TEXTLIST AUTOMATA_lepesek2
  0 = 'Készenléti állapot'
  1 = 'A szán indítása'
  3 = '6. hegesztés, várakozás a szánra'
  4 = '6. hegesztés, fej indítása'
  5 = '6. hegesztés, várakozás a fejre'
  6 = '6. hegesztés, hegesztés folyamatban'
  7 = '6. hegesztés, fej vissza'
  8 = '6. hegesztés, fej vissza'
  9 = 'A szán indítása'
  11 = '7. hegesztés, várakozás a szánra'
  12 = '7. hegesztés, fej indítása'
  13 = '7. hegesztés, várakozás a fejre'
  14 = '7. hegesztés, hegesztés folyamatban'
  15 = '7. hegesztés, fej vissza'
  16 = '7. hegesztés, fej vissza'
  17 = 'A szán indítása'
  18 = 'Kappe felhelyezés, várakozás a szánra'
  19 = 'Várakozás a robotra'
  20 = 'A robot eredmény törlésére vár'
  21 = 'A robot felhelyezi a kappét'
  22 = 'A szán indítása'
  23 = 'Kappe rögzítés, várakozás a szánra'
  24 = 'Kappe rögzítés indítása'
  27 = 'Várakozás a kappe rögzítés végére'
  28 = 'Mérés, várakozás a szánra'
  29 = 'Mérésválasztás'
  30 = 'Várakozás a mérés végére'
  31 = 'Lézeres jelölés előkészítése'
  32 = 'Várakozás a lézerre'
  33 = 'Lézertakaró nyitása'
  34 = 'Lézeres jelölés folyamatban'
  35 = 'Lézerezés állapot lekérdezés'
  36 = 'Lézerezés állapot lekérdezés'
  37 = 'Lézerezés állapot lekérdezés'
  40 = 'Lézertakaró zárása'
  41 = 'Kódellenörzés, várakozás a szánra'
  42 = 'Kódellenörzés folyamatban'
  43 = 'Kódellenörzés folyamatban'
  60 = 'Kiértékelés'
  99 = 'STOP utáni várakozás'
  100 = 'A szán indítása a szervízboxhoz'
  101 = 'Szervízbox, várakozás a szánra'
  103 = 'Várakozás az adapter\nkivételére'
  104 = 'Várakozás az adapter\nkivétele után'
  105 = 'Hegesztési hiba utáni várakozás'
  110 = 'A szán indítása a szervízboxhoz'
  111 = 'Várakozás a szánra és a folytatásra'
  112 = 'Várakozás a végmérőre, szán indítása'
  120 = 'Adapter pótlólagos felhelyezése'
  130 = 'Elhárítandó lézerhiba'
  140 = 'A szán indítása a szervízboxhoz'
  141 = 'Fedél megigazítására vár'
  142 = 'Kappe felhelyezés, várakozás a szánra'
  143 = 'Kappe felhelyezés indítása'
  150 = 'A szán indítása a szervízboxhoz'
  151 = 'Kappe pótlólagos felrakására vár'
  152 = 'Kappe felhelyezés, várakozás a szánra'
  153 = 'Kappe felhelyezés indítása'
  160 = 'Logolás hiba, várakozás a "Tovább" gombra.'
  170 = 'Várakozás folytatásra'
  171 = 'Hibás termék elengedése'
  180 = 'A szán a szervízboxhoz jön'
  181 = 'A "Tovább" gombra vár'
  200 = 'Pt tengely leállítása'
  201 = 'Hegesztés leállítása'
  202 = 'Hegesztö hibatörlés ellenörzése'
  203 = 'Sikertelen hegesztö hibatörlés\nutáni várakozás'
  204 = 'Várakozás a hegesztöfej\nvisszahúzódására'
  205 = 'Robot pozíció ellenörzése'
  206 = 'Robot HOME-ba érkezésére vár'
  207 = 'Végmérö RESET-elése'
  208 = 'Kappe RESET-elése'
  209 = 'Kappe RESET-elése'
  212 = 'Várakozás a végmérö, a lézer takaró lemez\nés a hegezstöfej alapállapotára'
  300 = 'Pt oldali folyamat felfüggesztve'
  400 = 'Kamera indítás'
  401 = 'Kamera kiértékelés'
  402 = 'Következö engedélyezett\nmüvelethez indul'
  410 = 'Várakozás a szánra ill. a\nfolytatásra'
  190 = 'A szán indítása a szervízboxhoz'
  191 = 'Szervízbox, várakozás a szánra'
  192 = 'A "Tovább" gombra vár'
  500 = 'Csatlakozó érzékeléshez'
  501 = 'Csatlakozó érzékelés indul'
  502 = 'Csatlakozó érzékelés kiértékelés'
  503 = 'A szán indítása'
  210 = 'Himba RESET-elése'
  211 = 'Himba RESET-elése'
   = ''
END_TEXTLIST

(* stored: Version 1.1.0.1, ProductVersion 3.1.4020.12
   TextList AUTOMATA_lepesek2: Id {c640c90e-3205-429a-9dab-fda536386133} *)
